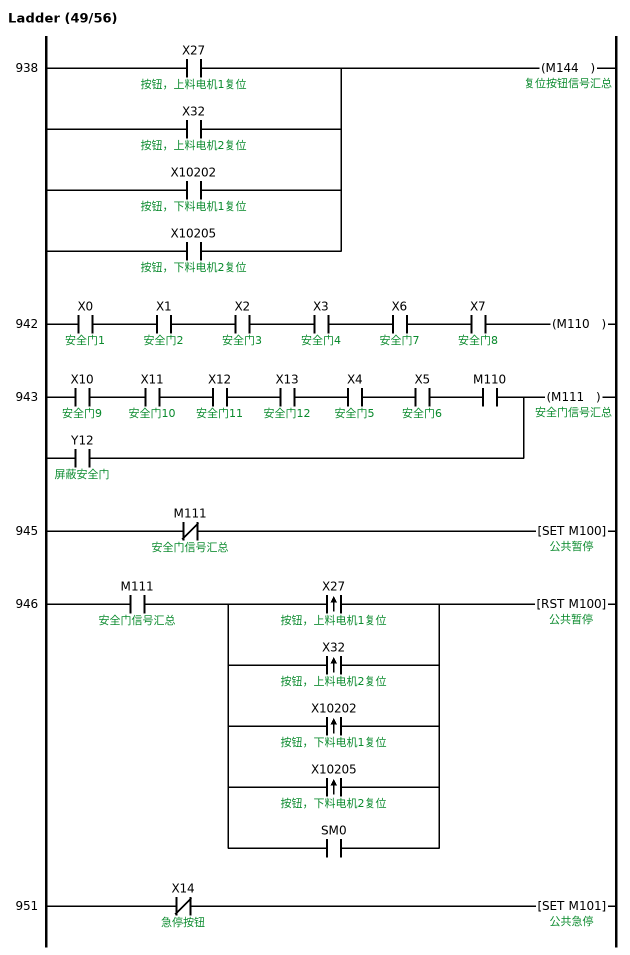
[picture p48: Ladder rows 938-951]
LD     X27	; 按钮，上料电机1复位
OR     X32	; 按钮，上料电机2复位
OR     X10202	; 按钮，下料电机1复位
OR     X10205	; 按钮，下料电机2复位
OUT    M144	; 复位按钮信号汇总
LD     X0	; 安全门1
AND    X1	; 安全门2
AND    X2	; 安全门3
AND    X3	; 安全门4
AND    X6	; 安全门7
AND    X7	; 安全门8
OUT    M110
LD     X10	; 安全门9
AND    X11	; 安全门10
AND    X12	; 安全门11
AND    X13	; 安全门12
AND    X4	; 安全门5
AND    X5	; 安全门6
AND    M110
OR     Y12	; 屏蔽安全门
OUT    M111	; 安全门信号汇总
LDI    M111	; 安全门信号汇总
SET    M100	; 公共暂停
LD     M111	; 安全门信号汇总
LDP    X27	; 按钮，上料电机1复位
ORP    X32	; 按钮，上料电机2复位
ORP    X10202	; 按钮，下料电机1复位
ORP    X10205	; 按钮，下料电机2复位
OR     SM0
ANB
RST    M100	; 公共暂停
LDI    X14	; 急停按钮
SET    M101	; 公共急停

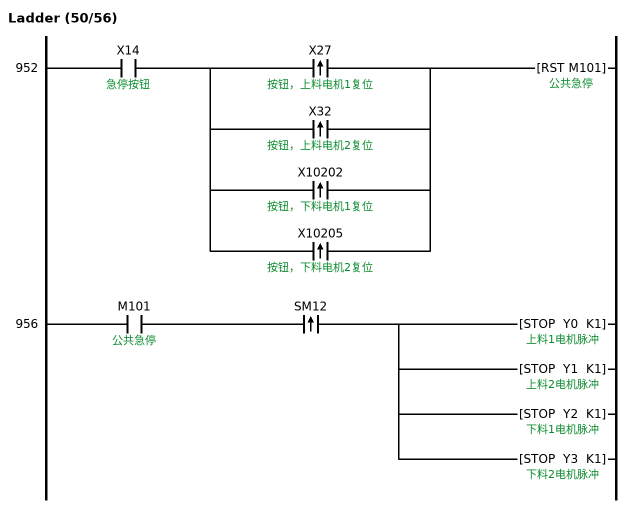
LD     X14	; 急停按钮
LDP    X27	; 按钮，上料电机1复位
ORP    X32	; 按钮，上料电机2复位
ORP    X10202	; 按钮，下料电机1复位
ORP    X10205	; 按钮，下料电机2复位
ANB
RST    M101	; 公共急停
LD     M101	; 公共急停
ANDP   SM12
STOP   Y0 K1	; 上料1电机脉冲
STOP   Y1 K1	; 上料2电机脉冲
STOP   Y2 K1	; 下料1电机脉冲
STOP   Y3 K1	; 下料2电机脉冲

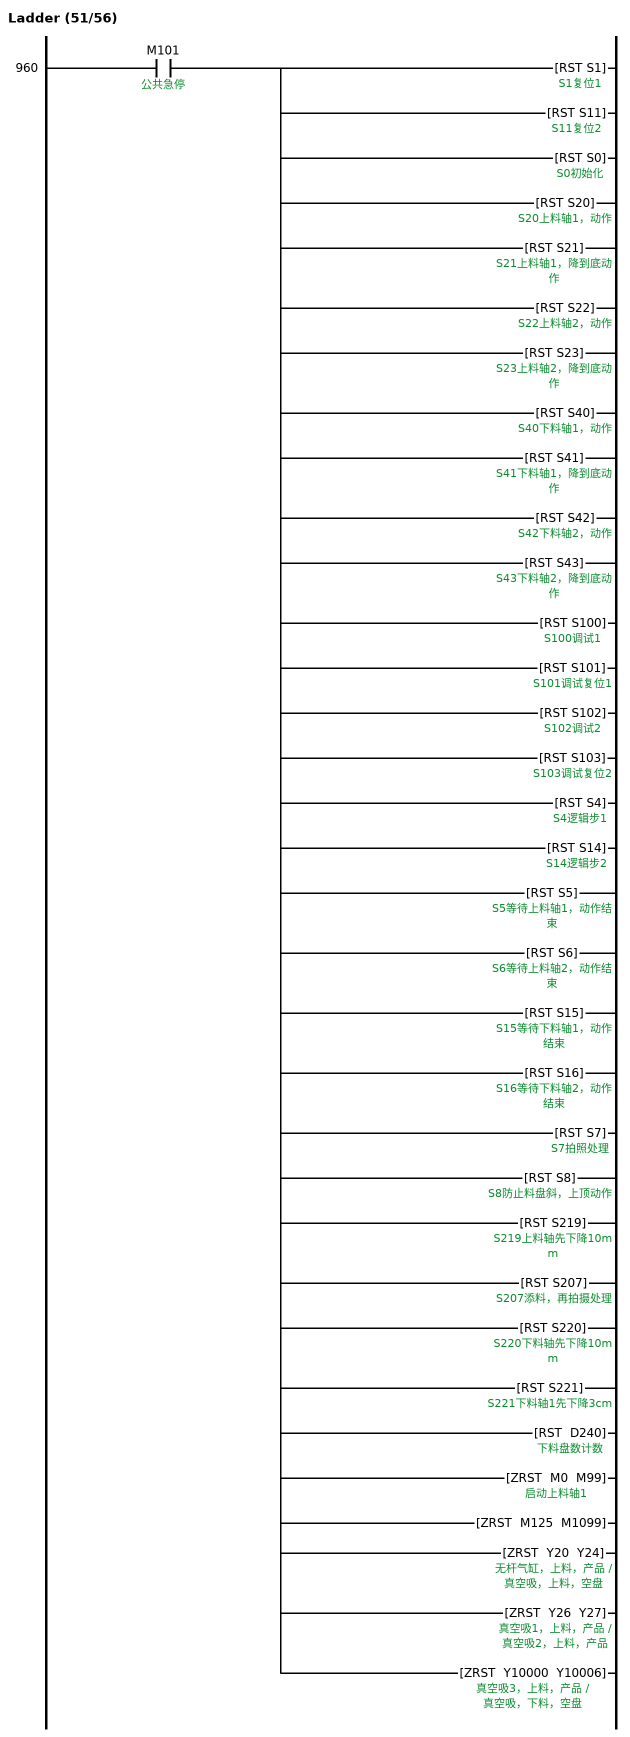
LD     M101	; 公共急停
RST    S1	; S1复位1
RST    S11	; S11复位2
RST    S0	; S0初始化
RST    S20	; S20上料轴1，动作
RST    S21	; S21上料轴1，降到底动作
RST    S22	; S22上料轴2，动作
RST    S23	; S23上料轴2，降到底动作
RST    S40	; S40下料轴1，动作
RST    S41	; S41下料轴1，降到底动作
RST    S42	; S42下料轴2，动作
RST    S43	; S43下料轴2，降到底动作
RST    S100	; S100调试1
RST    S101	; S101调试复位1
RST    S102	; S102调试2
RST    S103	; S103调试复位2
RST    S4	; S4逻辑步1
RST    S14	; S14逻辑步2
RST    S5	; S5等待上料轴1，动作结束
RST    S6	; S6等待上料轴2，动作结束
RST    S15	; S15等待下料轴1，动作结束
RST    S16	; S16等待下料轴2，动作结束
RST    S7	; S7拍照处理
RST    S8	; S8防止料盘斜，上顶动作
RST    S219	; S219上料轴先下降10mm
RST    S207	; S207添料，再拍摄处理
RST    S220	; S220下料轴先下降10mm
RST    S221	; S221下料轴1先下降3cm
RST    D240	; 下料盘数计数
ZRST   M0 M99	; 启动上料轴1
ZRST   M125 M1099
ZRST   Y20 Y24	; 无杆气缸，上料，产品 / 真空吸，上料，空盘
ZRST   Y26 Y27	; 真空吸1，上料，产品 / 真空吸2，上料，产品
ZRST   Y10000 Y10006	; 真空吸3，上料，产品 / 真空吸，下料，空盘

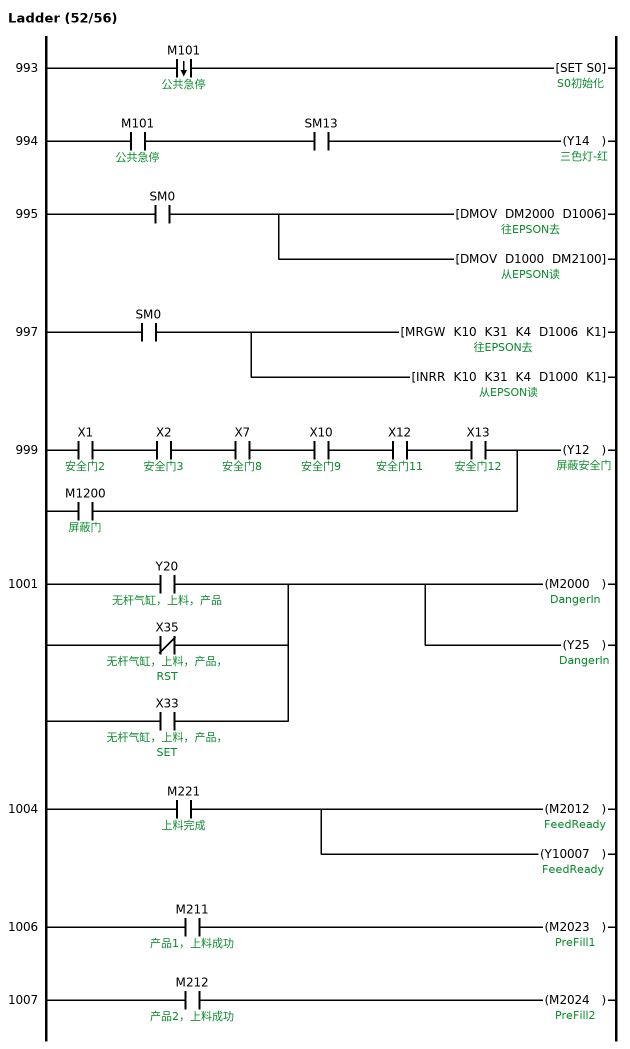
LDF    M101	; 公共急停
SET    S0	; S0初始化
LD     M101	; 公共急停
AND    SM13
OUT    Y14	; 三色灯-红
LD     SM0
DMOV   DM2000 D1006	; 往EPSON去
DMOV   D1000 DM2100	; 从EPSON读
LD     SM0
MRGW   K10 K31 K4 D1006 K1	; 往EPSON去
INRR   K10 K31 K4 D1000 K1	; 从EPSON读
LD     X1	; 安全门2
AND    X2	; 安全门3
AND    X7	; 安全门8
AND    X10	; 安全门9
AND    X12	; 安全门11
AND    X13	; 安全门12
OR     M1200	; 屏蔽门
OUT    Y12	; 屏蔽安全门
LD     Y20	; 无杆气缸，上料，产品
ORI    X35	; 无杆气缸，上料，产品，RST
OR     X33	; 无杆气缸，上料，产品，SET
OUT    M2000	; DangerIn
OUT    Y25	; DangerIn
LD     M221	; 上料完成
OUT    M2012	; FeedReady
OUT    Y10007	; FeedReady
LD     M211	; 产品1，上料成功
OUT    M2023	; PreFill1
LD     M212	; 产品2，上料成功
OUT    M2024	; PreFill2

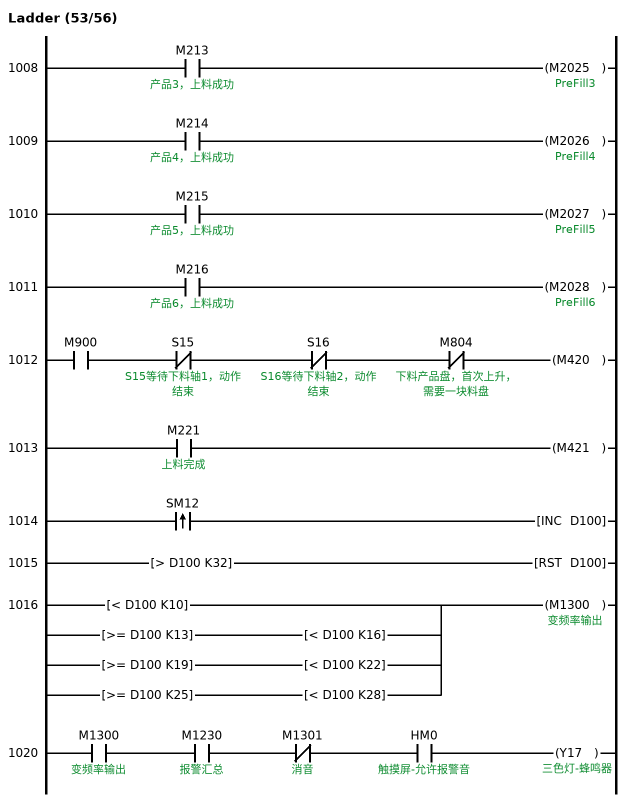
LD     M213	; 产品3，上料成功
OUT    M2025	; PreFill3
LD     M214	; 产品4，上料成功
OUT    M2026	; PreFill4
LD     M215	; 产品5，上料成功
OUT    M2027	; PreFill5
LD     M216	; 产品6，上料成功
OUT    M2028	; PreFill6
LD     M900
ANI    S15	; S15等待下料轴1，动作结束
ANI    S16	; S16等待下料轴2，动作结束
ANI    M804	; 下料产品盘，首次上升，需要一块料盘
OUT    M420
LD     M221	; 上料完成
OUT    M421
LDP    SM12
INC    D100
LD>    D100 K32
RST    D100
LD<    D100 K10
LD>=   D100 K13
AND<   D100 K16
ORB
LD>=   D100 K19
AND<   D100 K22
ORB
LD>=   D100 K25
AND<   D100 K28
ORB
OUT    M1300	; 变频率输出
LD     M1300	; 变频率输出
AND    M1230	; 报警汇总
ANI    M1301	; 消音
AND    HM0	; 触摸屏-允许报警音
OUT    Y17	; 三色灯-蜂鸣器

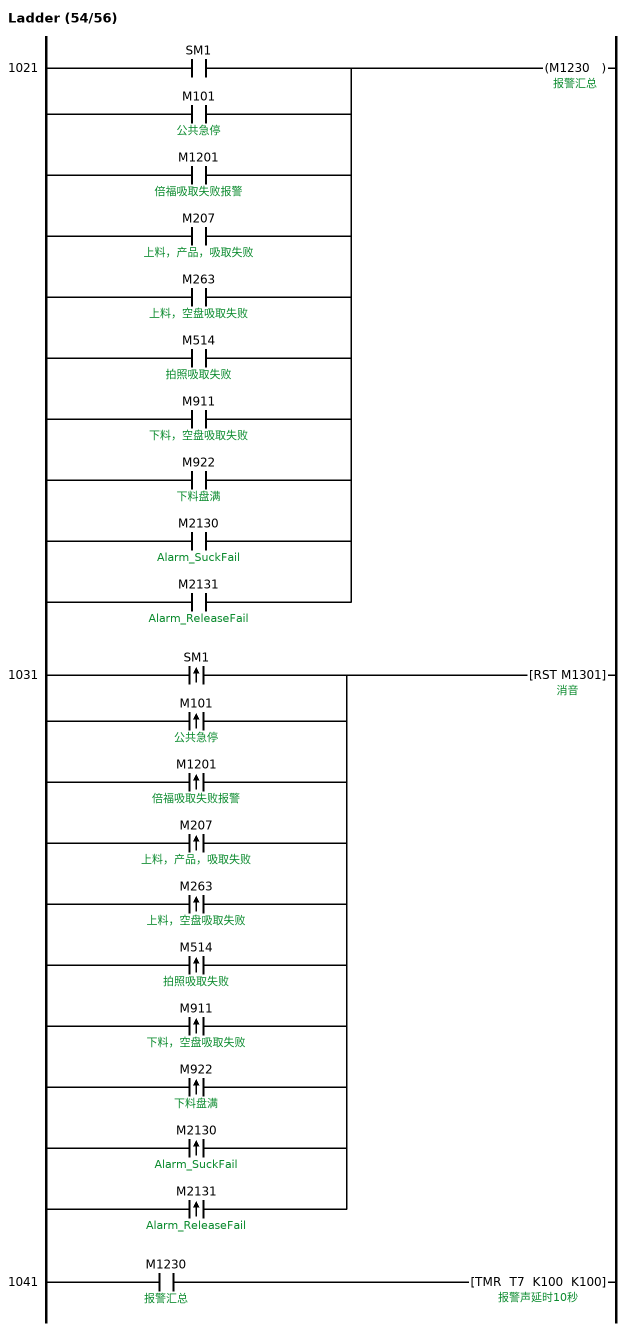
LD     SM1
OR     M101	; 公共急停
OR     M1201	; 倍福吸取失败报警
OR     M207	; 上料，产品，吸取失败
OR     M263	; 上料，空盘吸取失败
OR     M514	; 拍照吸取失败
OR     M911	; 下料，空盘吸取失败
OR     M922	; 下料盘满
OR     M2130	; Alarm_SuckFail
OR     M2131	; Alarm_ReleaseFail
OUT    M1230	; 报警汇总
LDP    SM1
ORP    M101	; 公共急停
ORP    M1201	; 倍福吸取失败报警
ORP    M207	; 上料，产品，吸取失败
ORP    M263	; 上料，空盘吸取失败
ORP    M514	; 拍照吸取失败
ORP    M911	; 下料，空盘吸取失败
ORP    M922	; 下料盘满
ORP    M2130	; Alarm_SuckFail
ORP    M2131	; Alarm_ReleaseFail
RST    M1301	; 消音
LD     M1230	; 报警汇总
TMR    T7 K100 K100	; 报警声延时10秒

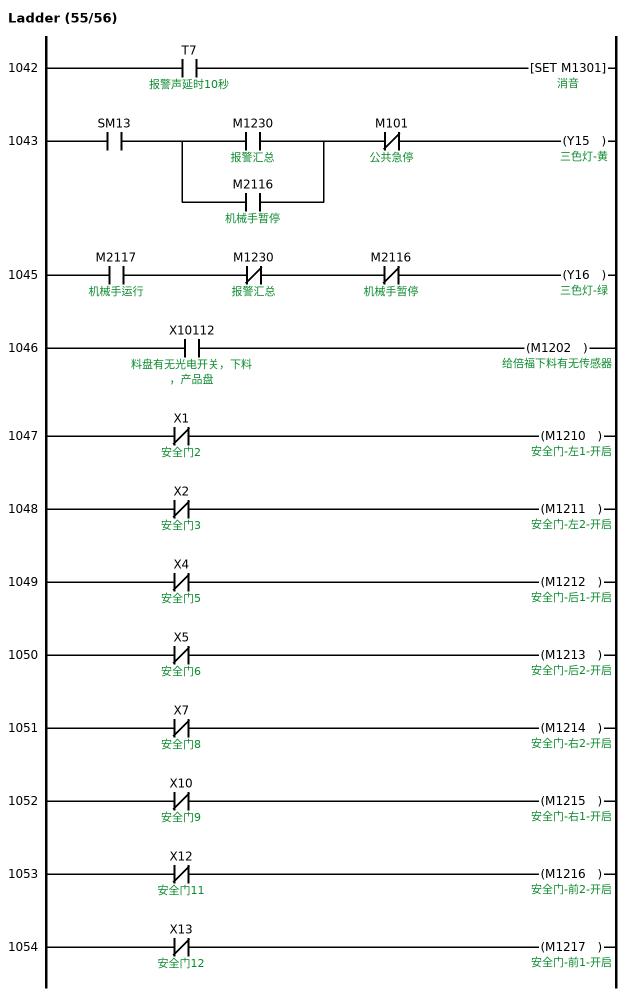
LD     T7	; 报警声延时10秒
SET    M1301	; 消音
LD     SM13
LD     M1230	; 报警汇总
OR     M2116	; 机械手暂停
ANB
ANI    M101	; 公共急停
OUT    Y15	; 三色灯-黄
LD     M2117	; 机械手运行
ANI    M1230	; 报警汇总
ANI    M2116	; 机械手暂停
OUT    Y16	; 三色灯-绿
LD     X10112	; 料盘有无光电开关，下料，产品盘
OUT    M1202	; 给倍福下料有无传感器
LDI    X1	; 安全门2
OUT    M1210	; 安全门-左1-开启
LDI    X2	; 安全门3
OUT    M1211	; 安全门-左2-开启
LDI    X4	; 安全门5
OUT    M1212	; 安全门-后1-开启
LDI    X5	; 安全门6
OUT    M1213	; 安全门-后2-开启
LDI    X7	; 安全门8
OUT    M1214	; 安全门-右2-开启
LDI    X10	; 安全门9
OUT    M1215	; 安全门-右1-开启
LDI    X12	; 安全门11
OUT    M1216	; 安全门-前2-开启
LDI    X13	; 安全门12
OUT    M1217	; 安全门-前1-开启

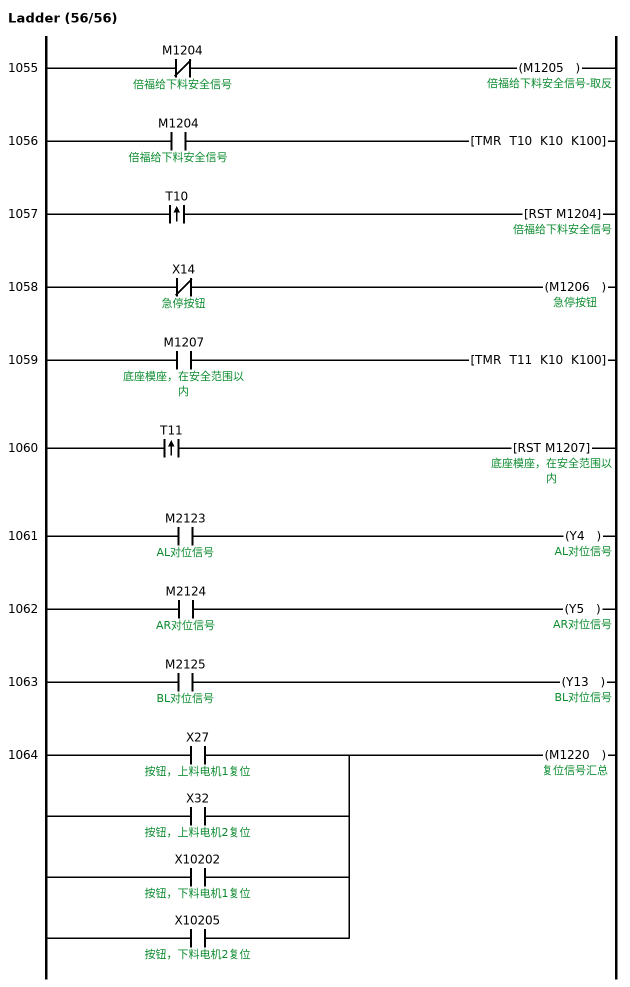
LDI    M1204	; 倍福给下料安全信号
OUT    M1205	; 倍福给下料安全信号-取反
LD     M1204	; 倍福给下料安全信号
TMR    T10 K10 K100
LDP    T10
RST    M1204	; 倍福给下料安全信号
LDI    X14	; 急停按钮
OUT    M1206	; 急停按钮
LD     M1207	; 底座模座，在安全范围以内
TMR    T11 K10 K100
LDP    T11
RST    M1207	; 底座模座，在安全范围以内
LD     M2123	; AL对位信号
OUT    Y4	; AL对位信号
LD     M2124	; AR对位信号
OUT    Y5	; AR对位信号
LD     M2125	; BL对位信号
OUT    Y13	; BL对位信号
LD     X27	; 按钮，上料电机1复位
OR     X32	; 按钮，上料电机2复位
OR     X10202	; 按钮，下料电机1复位
OR     X10205	; 按钮，下料电机2复位
OUT    M1220	; 复位信号汇总

COMMENTS (devices not used above)
X41	上下气缸，上料，产品，SET
X43	上下气缸，上料，空盘，SET
X10105	无杆气缸，下料，空盘，MID
X10107	上下气缸，下料，空盘，SET
X10210	上料吸盘光纤1
X10211	上料吸盘光纤2
X10212	下料吸盘光纤1
X10213	下料吸盘光纤2
M175	上料轴1，准备好
M176	上料轴2，准备好
M177	上料轴1，新上料
M201	上料命令
M218	等待上下气缸，上料，产品，复位到位
M243	报警：上料，缺料
M261	报警：空盘满，需要取走空盘
M272	报警：上料缺料
M2100	DangerOut
M2102	FeedEmpty
M2104	旋转气缸SET
S30	S30上料，运产品，动作
T0	上料，轴1，上到位延时